{attribute 'GeneratedUsingTerminal: EK1122-0000-0018'}
{attribute addProperty BoxType "EK1122-0000-0018"}
{attribute addProperty Id "Beckhoff_EPP5xxxsub_EK1100EK1100_1FC0878B2A_0001_EPP5001_0002_0016EPP5001_0B28D08722A_0002_EPP5101_0002_0016EPP5101_87AC78CF32A_0003_EPP5101_0002_0017EPP5101_87AC78CF32A_0004_EPP5101_0011_0016EPP5101_7476E94838A_0005_EPP5101_0011_0017EPP5101_7476E94838A_0006_EPP5101_1002_0016EPP5101_87AC78CF32A_0007_EPP5101_1002_0017EPP5101_87AC78CF32A_0008_EPP5151_0002_0016EPP5151_7476E94838A_0009_EPP5151_0002_0017EPP5151_7476E94838"}
{attribute addProperty CRC "4011796510"}
{attribute addProperty Size "304"}
TYPE Beckhoff_EPP5xxxEK1122_EF1F281E EXTENDS EK1122_1FC0878B :
STRUCT
	{attribute addProperty Name "Beckhoff EPP5xxxsub EK1100"}
	{attribute addProperty PreviousPort "Beckhoff EPP5xxxEK1122 : D"}
	Beckhoff_EPP5xxxsub_EK1100 : EK1100_1FC0878B;
	{attribute addProperty Name "A_0001(EPP5001-0002-0016)"}
	{attribute addProperty PreviousPort "Beckhoff EPP5xxxsub EK1100 : C"}
	A_0001_EPP5001_0002_0016 : EPP5001_0B28D087;
	{attribute addProperty Name "A_0002(EPP5101-0002-0016)"}
	{attribute addProperty PreviousPort "A_0001(EPP5001-0002-0016) : B"}
	A_0002_EPP5101_0002_0016 : EPP5101_87AC78CF;
	{attribute addProperty Name "A_0003(EPP5101-0002-0017)"}
	{attribute addProperty PreviousPort "A_0002(EPP5101-0002-0016) : B"}
	A_0003_EPP5101_0002_0017 : EPP5101_87AC78CF;
	{attribute addProperty Name "A_0004(EPP5101-0011-0016)"}
	{attribute addProperty PreviousPort "A_0003(EPP5101-0002-0017) : B"}
	A_0004_EPP5101_0011_0016 : EPP5101_7476E948;
	{attribute addProperty Name "A_0005(EPP5101-0011-0017)"}
	{attribute addProperty PreviousPort "A_0004(EPP5101-0011-0016) : B"}
	A_0005_EPP5101_0011_0017 : EPP5101_7476E948;
	{attribute addProperty Name "A_0006(EPP5101-1002-0016)"}
	{attribute addProperty PreviousPort "A_0005(EPP5101-0011-0017) : B"}
	A_0006_EPP5101_1002_0016 : EPP5101_87AC78CF;
	{attribute addProperty Name "A_0007(EPP5101-1002-0017)"}
	{attribute addProperty PreviousPort "A_0006(EPP5101-1002-0016) : B"}
	A_0007_EPP5101_1002_0017 : EPP5101_87AC78CF;
	{attribute addProperty Name "A_0008(EPP5151-0002-0016)"}
	{attribute addProperty PreviousPort "A_0007(EPP5101-1002-0017) : B"}
	A_0008_EPP5151_0002_0016 : EPP5151_7476E948;
	{attribute addProperty Name "A_0009(EPP5151-0002-0017)"}
	{attribute addProperty PreviousPort "A_0008(EPP5151-0002-0016) : B"}
	A_0009_EPP5151_0002_0017 : EPP5151_7476E948;
END_STRUCT
END_TYPE

(* stored: Version 1.2.0.0, ProductVersion 3.1.4024.11
   DUT Beckhoff_EPP5xxxEK1122_EF1F281E: Id {9c37c80d-a8bd-4687-a308-ef356c516a37} *)
